// TIA Portal V20 export
DATA_BLOCK "BK04"   // DB193
// stored: MemoryReserve 100
   VAR
      "X10-1 SPLICING L-MODULE MOVER BACKWARD" : Bool;
      "X11-1 SPLICING R-MODULE MOVER BACKWARD" : Bool;
      "X12-1 ELECTRODE L-HOLDER MOVER FORWARD" : Bool;
      "X13-1 ELECTRODE R-HOLDER MOVER FORWARD" : Bool;
      "X14-1 TAPE LOADING TURN HOMING" : Bool;
      "X15-1 TAPE ATTACH UNIT BACKWARD" : Bool;
      "X16-1 TAPING VACUUM PRESSURE SWITCH" : Bool;
      "X17-1 SPARE" : Bool;
      "X10-2 SPLICING L-MODULE MOVER FORWARD" : Bool;
      "X11-2 SPLICING R-MODULE MOVER FORWARD" : Bool;
      "X12-2 ELECTRODE L-HOLDER MOVER BACKWARD" : Bool;
      "X13-2 ELECTRODE R-HOLDER MOVER BACKWARD" : Bool;
      "X14-2 TAPE LOADING TURN ROTATE" : Bool;
      "X15-2 TAPE ATTACH UNIT FORWARD" : Bool;
      "X16-2 SPARE" : Bool;
      "X17-2 SPARE" : Bool;
   END_VAR
BEGIN
END_DATA_BLOCK
